// TIA Portal V19 export
VAR_GLOBAL   // PLC tag table "Default tag table"
   Tag_1 AT %I0.0 : Bool;
   Tag_2 AT %Q0.0 : Bool;
END_VAR
